// Mitsubishi GX Works2 project: projectB   PLC: FX3G

// global labels: Global1
VAR_GLOBAL
  startDayButton AT X007 : BOOL;
  initialBiscuit AT D1100 : REAL;
END_VAR
VAR_GLOBAL CONSTANT
  min6 : REAL := 6;
END_VAR
VAR_GLOBAL
  EnoughBiscuit AT M0 : BOOL;
  initialChocolate AT D1102 : REAL;
END_VAR
VAR_GLOBAL CONSTANT
  min240 : REAL := 240;
END_VAR
VAR_GLOBAL
  EnoughChocolate AT M1 : BOOL;
  initialCream AT D1104 : REAL;
END_VAR
VAR_GLOBAL CONSTANT
  min300 : REAL := 300;
END_VAR
VAR_GLOBAL
  EnoughCream AT M2 : BOOL;
  InitialDay AT M60 : BOOL;
  storageBiscuit AT D1106 : REAL;
  storageChocolate AT D1108 : REAL;
  DayStarted AT M54 : BOOL;
  WorkingDay AT Y007 : BOOL;
  EnoughBiscuitForIteration AT M4 : BOOL;
  EnoughChoclateForIteration AT M5 : BOOL;
  EnoughCreamForIteration AT M6 : BOOL;
  EnoughStorage AT M100 : BOOL;
  PreperForPipe AT X011 : BOOL;
END_VAR
VAR_GLOBAL CONSTANT
  ThreeHoundred : REAL := 300;
END_VAR
VAR_GLOBAL
  PipingContainer AT D1112 : REAL;
END_VAR
VAR_GLOBAL CONSTANT
  Six : REAL := 6;
END_VAR
VAR_GLOBAL
  BiscuitBox AT D1114 : REAL;
  MoveCream AT M95 : BOOL;
  MoveBiscuit AT M94 : BOOL;
  startMachineA AT X010 : BOOL;
  MachineAWorking AT M96 : BOOL;
  BoxInPlace AT X001 : BOOL;
  TempartureIsOk AT M82 : BOOL;
  NoSignalHasSent AT X002 : BOOL;
  StopMachine AT X005 : BOOL;
  signalHasSent AT X002 : BOOL;
  Piping AT Y004 : BOOL;
  AnalogInput2 AT D8281 : INT;
  SaveTemp AT D1200 : REAL;
END_VAR
VAR_GLOBAL CONSTANT
  Ten : REAL := 10;
  Min15 : REAL := 15;
  Max30 : REAL := 30;
END_VAR
VAR_GLOBAL
  GoodTemp1 AT M80 : BOOL;
  GoodTemp2 AT M81 : BOOL;
  Timer1 AT TC1 : BOOL;
END_VAR
VAR_GLOBAL CONSTANT
  Timer40 : WORD := 40;
END_VAR
VAR_GLOBAL
  Temp60 AT M65 : BOOL;
  TimerFinished1 AT TS1 : BOOL;
  Lamp0 AT M62 : BOOL;
  Timer2 AT TC2 : BOOL;
  TimerFinished2 AT TS2 : BOOL;
  Lamp1 AT M63 : BOOL;
END_VAR
VAR_GLOBAL CONSTANT
  Timer10 : INT := 10;
END_VAR
VAR_GLOBAL
  startblinking AT M61 : BOOL;
  TimerMovingAB AT TC3 : BOOL;
  TimerFinished3 AT TS3 : BOOL;
  Lamp01 AT Y000 : BOOL;
  Lamp02 AT Y001 : BOOL;
  Temp65 AT M65 : BOOL;
  EndIteration AT M7 : BOOL;
  EndDay AT M101 : BOOL;
  Temp AT M40 : BOOL;
  FinaleBlink AT M66 : BOOL;
  StartCoating AT X006 : BOOL;
END_VAR
VAR_GLOBAL CONSTANT
  Above6 : REAL := 6;
  Under5 : REAL := 5;
END_VAR
VAR_GLOBAL
  AnalogInput1 AT D8280 : INT;
  DoubleCoating AT M20 : BOOL;
  SingleCoating AT M21 : BOOL;
END_VAR
VAR_GLOBAL CONSTANT
  Coat20 : REAL := 120;
  Coat40 : REAL := 240;
END_VAR
VAR_GLOBAL
  ChocolateContainer AT D1116 : REAL;
  MoveChocolate AT M23 : BOOL;
  TimerCoating AT TC4 : BOOL;
END_VAR
VAR_GLOBAL CONSTANT
  Timer50 : INT := 50;
END_VAR
VAR_GLOBAL
  TimerFinished4 AT TS4 : BOOL;
  Coating AT Y003 : BOOL;
  PackKrembo AT X000 : BOOL;
  CounterPacking AT CC1 : BOOL;
END_VAR
VAR_GLOBAL CONSTANT
  Counter5 : INT := 5;
END_VAR
VAR_GLOBAL
  Packing AT Y002 : BOOL;
  CounterFinished1 AT CS1 : BOOL;
  CounterPacking2 AT CC2 : BOOL;
END_VAR
VAR_GLOBAL CONSTANT
  Counter6 : INT := 6;
END_VAR
VAR_GLOBAL
  CounterFinished2 AT CS2 : BOOL;
  TimerEndDay AT TC6 : BOOL;
END_VAR
VAR_GLOBAL CONSTANT
  Timer30 : INT := 30;
END_VAR
VAR_GLOBAL
  TimerFinished6 AT TS6 : BOOL;
END_VAR
VAR_GLOBAL CONSTANT
  Count0 : REAL;
END_VAR
VAR_GLOBAL
  Krembos AT D1118 : REAL;
END_VAR
VAR_GLOBAL CONSTANT
  Constant6 : REAL := 6;
  Constant10 : REAL := 10;
END_VAR
VAR_GLOBAL
  InputForChocolate AT D1200 : REAL;
  ChocolateSaved AT M25 : BOOL;
  TempUnder30 AT X004 : BOOL;
  TempUnder15 AT X003 : BOOL;
END_VAR
VAR_GLOBAL CONSTANT
  Timer400 : WORD := 400;
END_VAR
VAR_GLOBAL
  xxx AT M300 : BOOL;
  StorageCream AT D1120 : REAL;
END_VAR
VAR_GLOBAL CONSTANT
  FourHundred : REAL := 400;
  Zero : REAL;
  Fourty : INT := 40;
END_VAR
VAR_GLOBAL
  ShowKrembos AT D1122 : REAL;
  AnalogOutput AT D8282 : INT;
  StopPiping AT M200 : BOOL;
  MovingFinished AT M201 : BOOL;
  Counter7 AT CC7 : BOOL;
END_VAR
VAR_GLOBAL CONSTANT
  Two : INT := 2;
END_VAR
VAR_GLOBAL
  CounterFinisher7 AT CS7 : BOOL;
  Counter8 AT CC8 : BOOL;
END_VAR
VAR_GLOBAL CONSTANT
  Three : INT := 3;
END_VAR
VAR_GLOBAL
  CoatingFinished AT M202 : BOOL;
  CounterFinished8 AT CS8 : BOOL;
END_VAR
VAR_GLOBAL CONSTANT
  One : INT := 1;
END_VAR
VAR_GLOBAL
  Counter9 AT CC9 : BOOL;
  PipingFinished AT M203 : BOOL;
  CounterFinished9 AT CS9 : BOOL;
END_VAR

// task Task_01 (event TRUE, interval 0, priority 31): POU_01

PROGRAM POU_01
(* structured ladder/FBD written out as ST: instructions are called as NAME(EN, inputs, outputs); _pN, _eN, _tN stand for wires *)
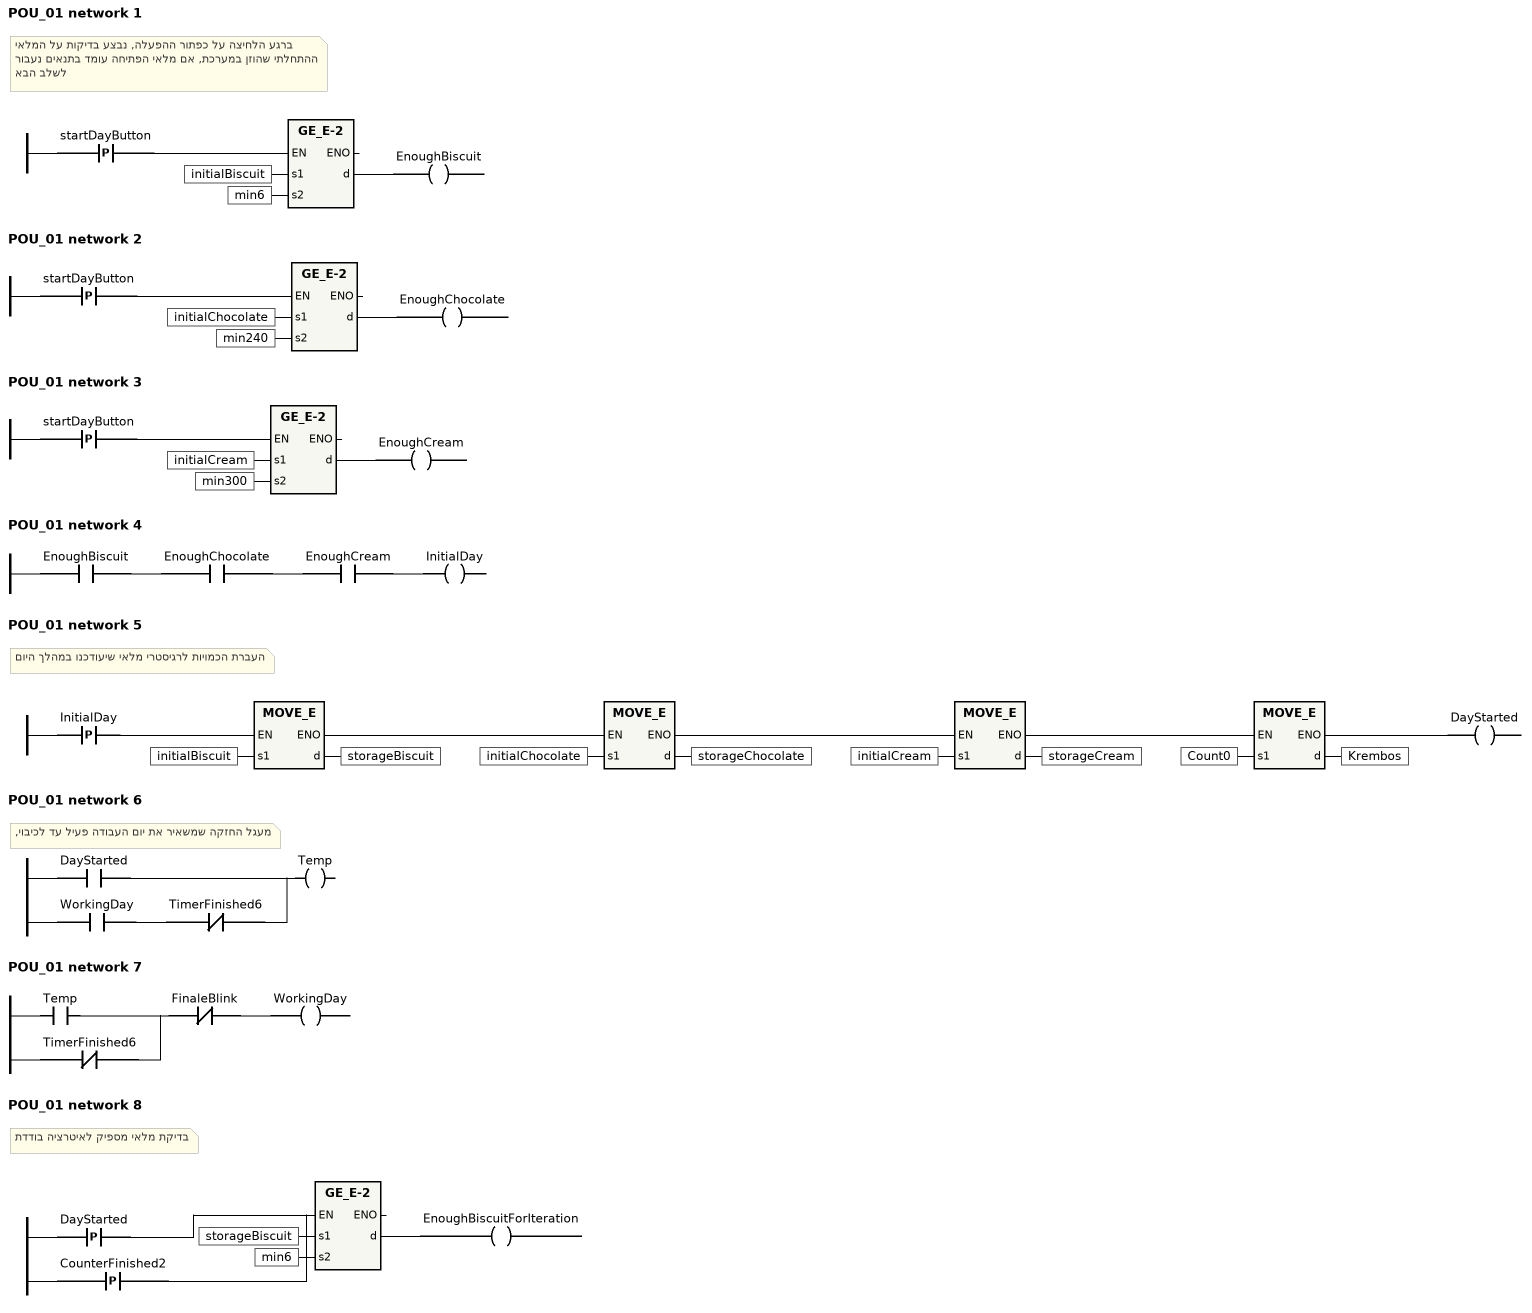
(* network 1 *)
(* ברגע הלחיצה על כפתור ההפעלה, נבצע בדיקות על המלאי ההתחלתי שהוזן במערכת, אם מלאי הפתיחה עומד בתנאים נעבור לשלב הבא *)
GE_E(LDP(TRUE, startDayButton), initialBiscuit, min6, _t1);
EnoughBiscuit := _t1;
(* network 2 *)
GE_E(LDP(TRUE, startDayButton), initialChocolate, min240, _t1);
EnoughChocolate := _t1;
(* network 3 *)
GE_E(LDP(TRUE, startDayButton), initialCream, min300, _t1);
EnoughCream := _t1;
(* network 4 *)
InitialDay := EnoughBiscuit AND EnoughChocolate AND EnoughCream;
(* network 5 *)
(* העברת הכמויות לרגיסטרי מלאי שיעודכנו במהלך היום *)
_e1 := MOVE_E(LDP(TRUE, InitialDay), initialBiscuit, storageBiscuit);
_e2 := MOVE_E(_e1, initialChocolate, storageChocolate);
_e3 := MOVE_E(_e2, initialCream, storageCream);
_e4 := MOVE_E(_e3, Count0, Krembos);
DayStarted := _e4;
(* network 6 *)
(* מעגל החזקה שמשאיר את יום העבודה פעיל עד לכיבוי, *)
Temp := DayStarted OR (WorkingDay AND NOT TimerFinished6);
(* network 7 *)
WorkingDay := (Temp OR (NOT TimerFinished6)) AND NOT FinaleBlink;
(* network 8 *)
(* בדיקת מלאי מספיק לאיטרציה בודדת *)
GE_E(LDP(TRUE, DayStarted) OR LDP(TRUE, CounterFinished2), storageBiscuit, min6, _t1);
EnoughBiscuitForIteration := _t1;
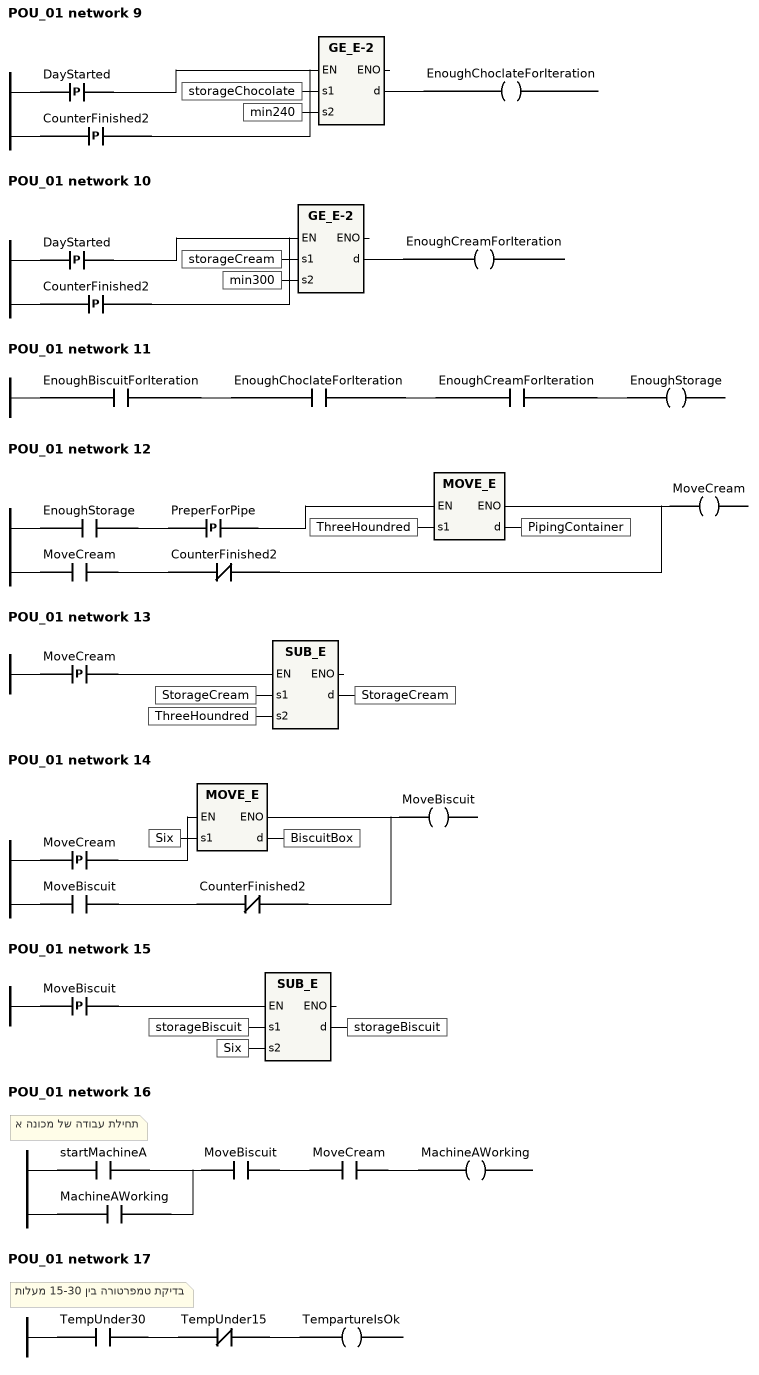
(* network 9 *)
GE_E(LDP(TRUE, DayStarted) OR LDP(TRUE, CounterFinished2), storageChocolate, min240, _t1);
EnoughChoclateForIteration := _t1;
(* network 10 *)
GE_E(LDP(TRUE, DayStarted) OR LDP(TRUE, CounterFinished2), storageCream, min300, _t1);
EnoughCreamForIteration := _t1;
(* network 11 *)
EnoughStorage := EnoughBiscuitForIteration AND EnoughChoclateForIteration AND EnoughCreamForIteration;
(* network 12 *)
_e1 := MOVE_E(EnoughStorage AND LDP(TRUE, PreperForPipe), ThreeHoundred, PipingContainer);
MoveCream := _e1 OR (MoveCream AND NOT CounterFinished2);
(* network 13 *)
SUB_E(LDP(TRUE, MoveCream), StorageCream, ThreeHoundred, StorageCream);
(* network 14 *)
_e1 := MOVE_E(LDP(TRUE, MoveCream), Six, BiscuitBox);
MoveBiscuit := _e1 OR (MoveBiscuit AND NOT CounterFinished2);
(* network 15 *)
SUB_E(LDP(TRUE, MoveBiscuit), storageBiscuit, Six, storageBiscuit);
(* network 16 *)
(* תחילת עבודה של מכונה א *)
MachineAWorking := ((startMachineA OR MachineAWorking) AND MoveBiscuit) AND MoveCream;
(* network 17 *)
(* בדיקת טמפרטורה בין 15-30 מעלות *)
TempartureIsOk := TempUnder30 AND NOT TempUnder15;
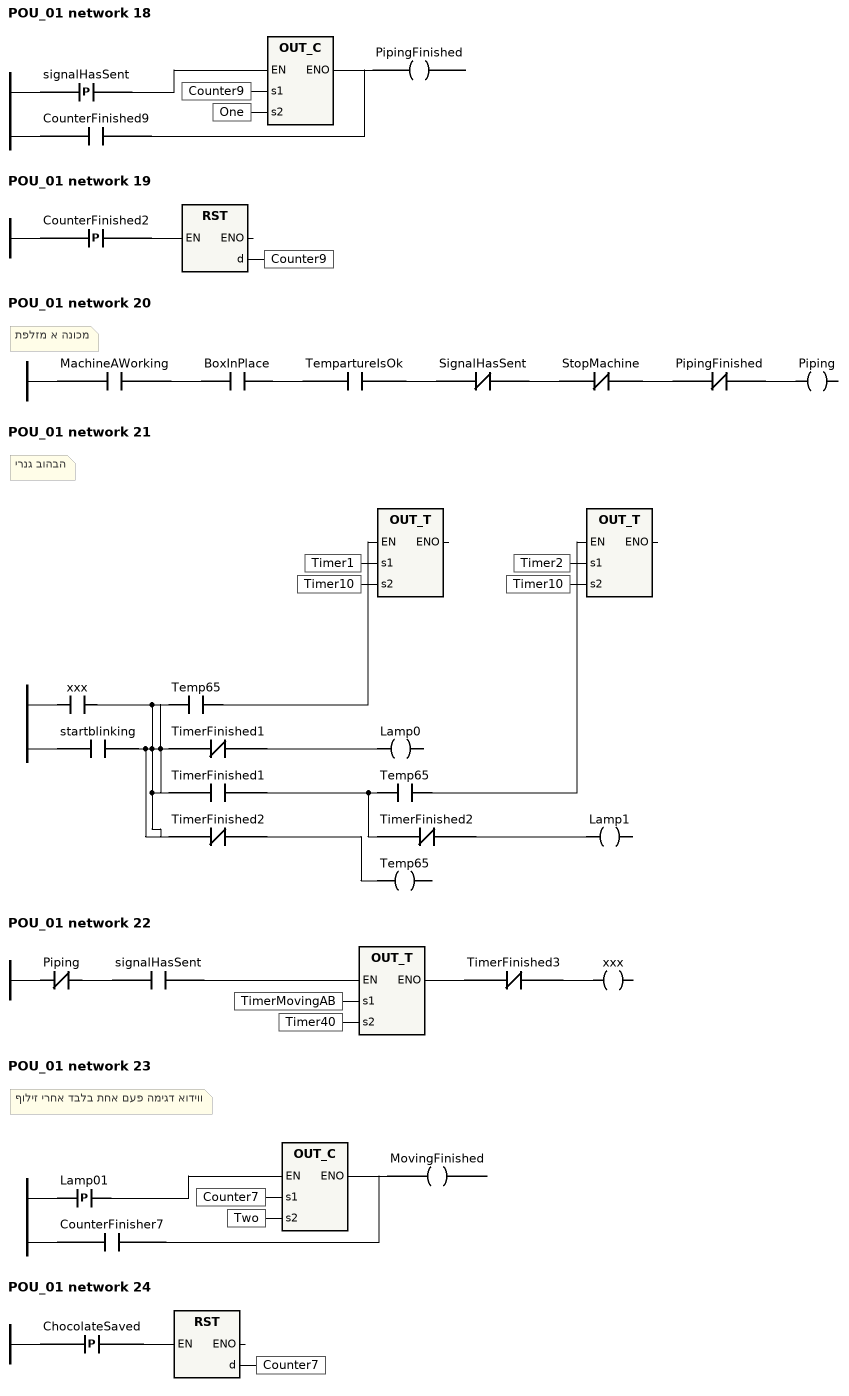
(* network 18 *)
_e1 := OUT_C(LDP(TRUE, signalHasSent), Counter9, One);
PipingFinished := _e1 OR CounterFinished9;
(* network 19 *)
RST(LDP(TRUE, CounterFinished2), Counter9);
(* network 20 *)
(* מכונה א מזלפת *)
Piping := MachineAWorking AND BoxInPlace AND TempartureIsOk AND NOT SignalHasSent AND NOT StopMachine AND NOT PipingFinished;
(* network 21 *)
(* הבהוב גנרי *)
_p1 := xxx OR startblinking;
OUT_T(_p1 AND Temp65, Timer1, Timer10);
Lamp0 := _p1 AND NOT TimerFinished1;
_p2 := _p1 AND TimerFinished1;
OUT_T(_p2 AND Temp65, Timer2, Timer10);
Lamp1 := _p2 AND NOT TimerFinished2;
Temp65 := _p1 AND NOT TimerFinished2;
(* network 22 *)
_e1 := OUT_T(NOT Piping AND signalHasSent, TimerMovingAB, Timer40);
xxx := _e1 AND NOT TimerFinished3;
(* network 23 *)
(* ווידוא דגימה פעם אחת בלבד אחרי זילוף *)
_e1 := OUT_C(LDP(TRUE, Lamp01), Counter7, Two);
MovingFinished := _e1 OR CounterFinisher7;
(* network 24 *)
RST(LDP(TRUE, ChocolateSaved), Counter7);
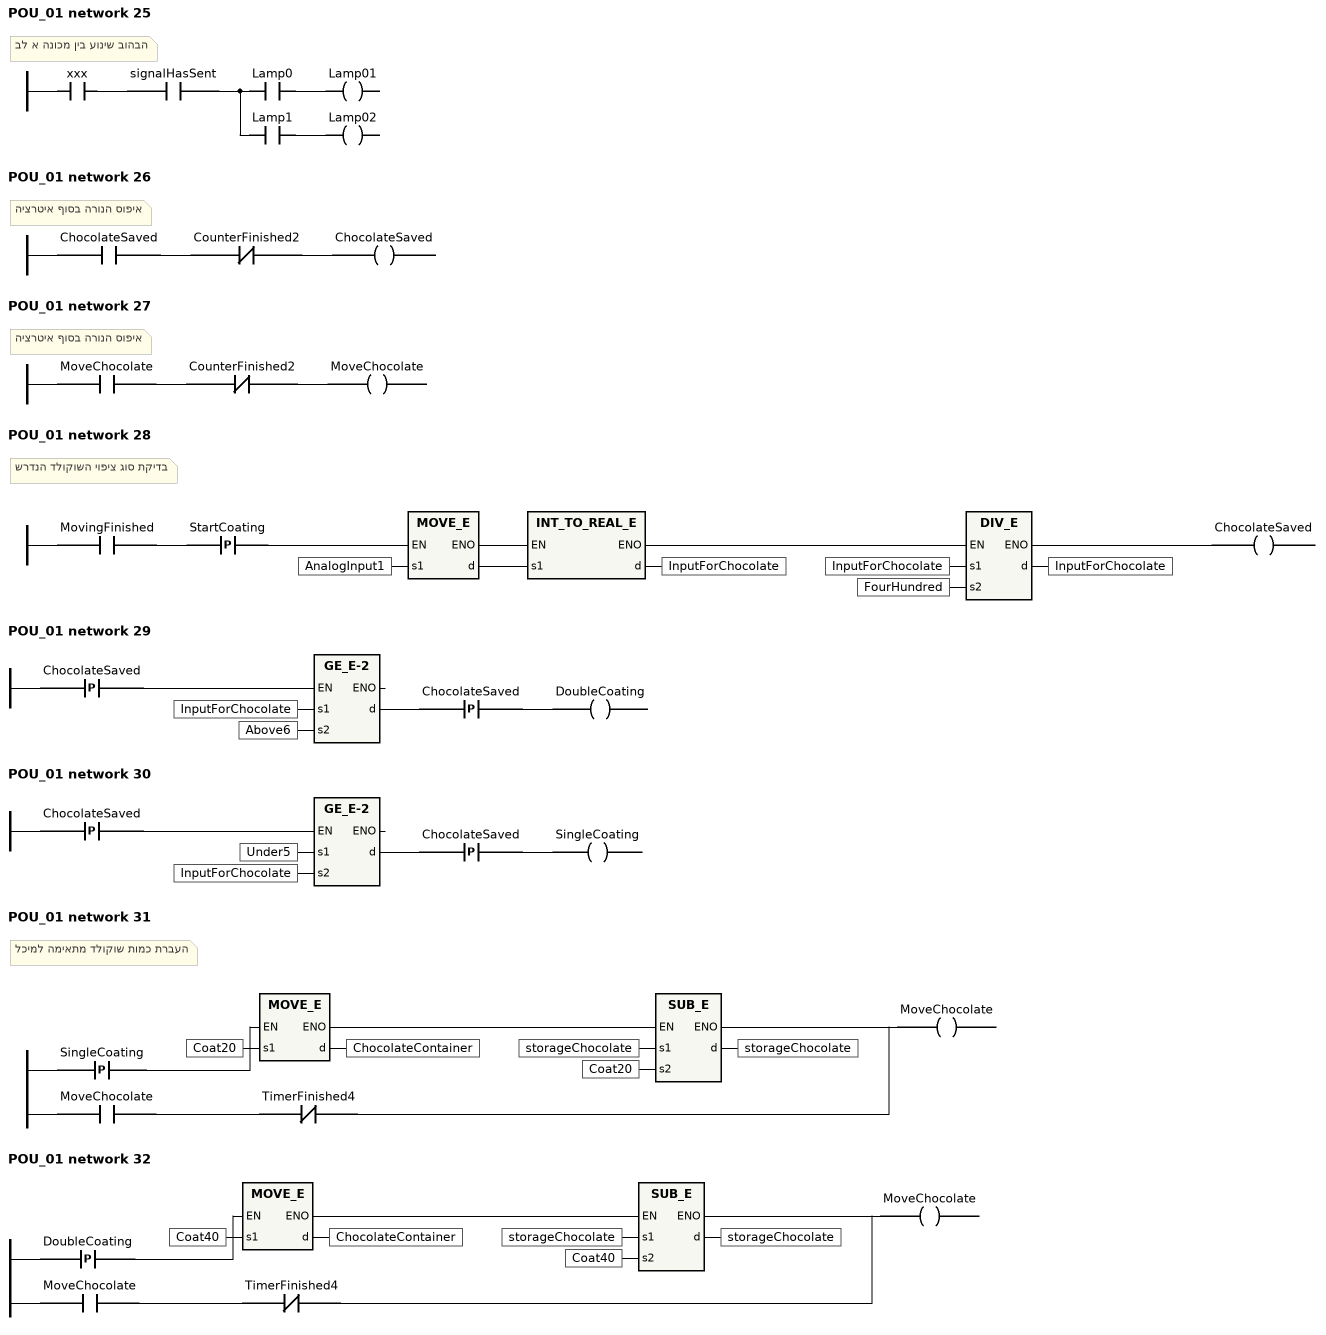
(* network 25 *)
(* הבהוב שינוע בין מכונה א לב *)
_p1 := xxx AND signalHasSent;
Lamp01 := _p1 AND Lamp0;
Lamp02 := _p1 AND Lamp1;
(* network 26 *)
(* איפוס הנורה בסוף איטרציה *)
ChocolateSaved := ChocolateSaved AND NOT CounterFinished2;
(* network 27 *)
(* איפוס הנורה בסוף איטרציה *)
MoveChocolate := MoveChocolate AND NOT CounterFinished2;
(* network 28 *)
(* בדיקת סוג ציפוי השוקולד הנדרש *)
_e2 := MOVE_E(MovingFinished AND LDP(TRUE, StartCoating), AnalogInput1, _t1);
_e3 := INT_TO_REAL_E(_e2, _t1, InputForChocolate);
_e4 := DIV_E(_e3, InputForChocolate, FourHundred, InputForChocolate);
ChocolateSaved := _e4;
(* network 29 *)
GE_E(LDP(TRUE, ChocolateSaved), InputForChocolate, Above6, _t1);
DoubleCoating := _t1 AND LDP(TRUE, ChocolateSaved);
(* network 30 *)
GE_E(LDP(TRUE, ChocolateSaved), Under5, InputForChocolate, _t1);
SingleCoating := _t1 AND LDP(TRUE, ChocolateSaved);
(* network 31 *)
(* העברת כמות שוקולד מתאימה למיכל *)
_e1 := MOVE_E(LDP(TRUE, SingleCoating), Coat20, ChocolateContainer);
_e2 := SUB_E(_e1, storageChocolate, Coat20, storageChocolate);
MoveChocolate := _e2 OR (MoveChocolate AND NOT TimerFinished4);
(* network 32 *)
_e1 := MOVE_E(LDP(TRUE, DoubleCoating), Coat40, ChocolateContainer);
_e2 := SUB_E(_e1, storageChocolate, Coat40, storageChocolate);
MoveChocolate := _e2 OR (MoveChocolate AND NOT TimerFinished4);
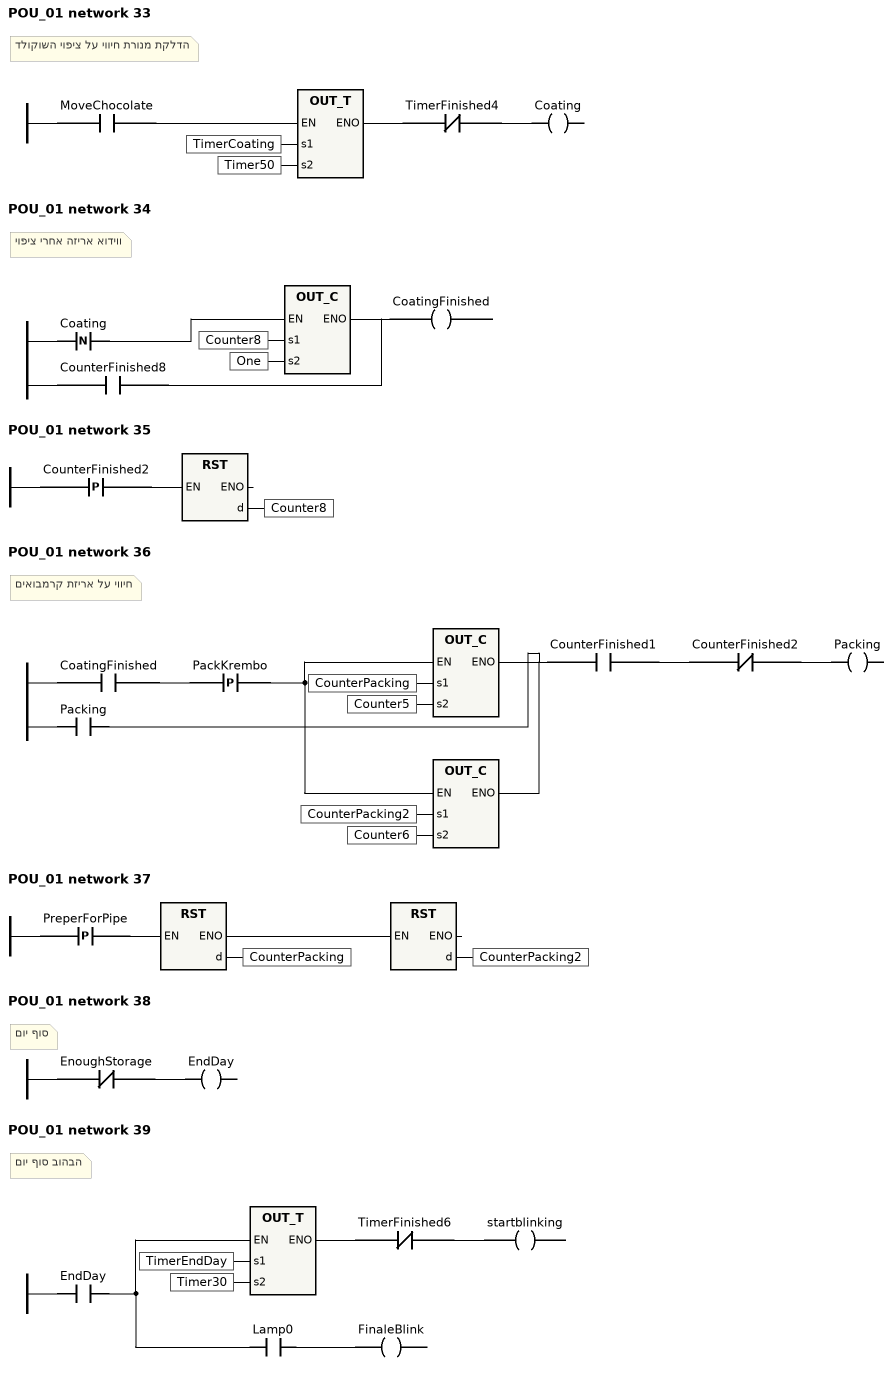
(* network 33 *)
(* הדלקת מנורת חיווי על ציפוי השוקולד *)
_e1 := OUT_T(MoveChocolate, TimerCoating, Timer50);
Coating := _e1 AND NOT TimerFinished4;
(* network 34 *)
(* ווידוא אריזה אחרי ציפוי *)
_e1 := OUT_C(LDF(TRUE, Coating), Counter8, One);
CoatingFinished := _e1 OR CounterFinished8;
(* network 35 *)
RST(LDP(TRUE, CounterFinished2), Counter8);
(* network 36 *)
(* חיווי על אריזת קרמבואים *)
_p1 := CoatingFinished AND LDP(TRUE, PackKrembo);
_e2 := OUT_C(_p1, CounterPacking, Counter5);
_e3 := OUT_C(_p1, CounterPacking2, Counter6);
Packing := ((_e2 OR _e3 OR Packing) AND CounterFinished1) AND NOT CounterFinished2;
(* network 37 *)
_e1 := RST(LDP(TRUE, PreperForPipe), CounterPacking);
RST(_e1, CounterPacking2);
(* network 38 *)
(* סוף יום *)
EndDay := NOT EnoughStorage;
(* network 39 *)
(* הבהוב סוף יום *)
_e1 := OUT_T(EndDay, TimerEndDay, Timer30);
startblinking := _e1 AND NOT TimerFinished6;
FinaleBlink := EndDay AND Lamp0;
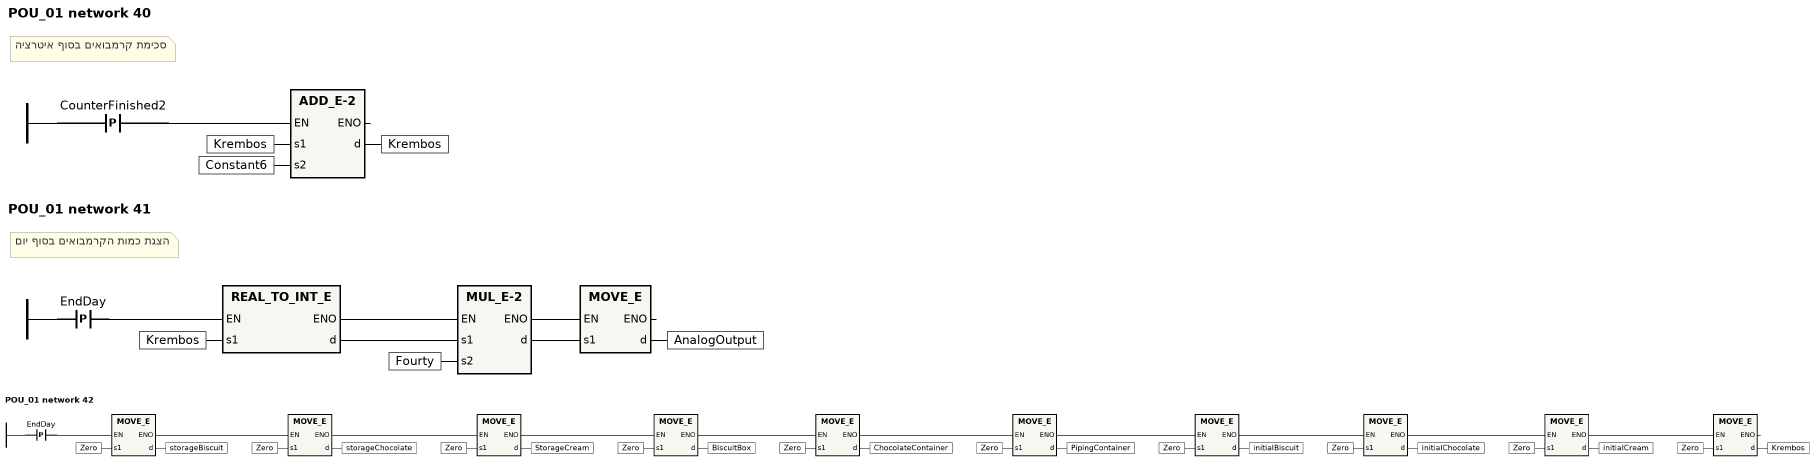
(* network 40 *)
(* סכימת קרמבואים בסוף איטרציה *)
ADD_E(LDP(TRUE, CounterFinished2), Krembos, Constant6, Krembos);
(* network 41 *)
(* הצגת כמות הקרמבואים בסוף יום *)
_e2 := REAL_TO_INT_E(LDP(TRUE, EndDay), Krembos, _t1);
_e4 := MUL_E(_e2, _t1, Fourty, _t3);
MOVE_E(_e4, _t3, AnalogOutput);
(* network 42 *)
_e1 := MOVE_E(LDP(TRUE, EndDay), Zero, storageBiscuit);
_e2 := MOVE_E(_e1, Zero, storageChocolate);
_e3 := MOVE_E(_e2, Zero, StorageCream);
_e4 := MOVE_E(_e3, Zero, BiscuitBox);
_e5 := MOVE_E(_e4, Zero, ChocolateContainer);
_e6 := MOVE_E(_e5, Zero, PipingContainer);
_e7 := MOVE_E(_e6, Zero, initialBiscuit);
_e8 := MOVE_E(_e7, Zero, initialChocolate);
_e9 := MOVE_E(_e8, Zero, initialCream);
MOVE_E(_e9, Zero, Krembos);
END_PROGRAM
